// TIA Portal V20 export
FUNCTION_BLOCK "CallProcessCount"   // FB2, LAD
// stored: MemoryReserve 100, SetENOAutomatically false
   VAR
      statPulse { ExternalAccessible := 'False'; ExternalVisible := 'False'; ExternalWritable := 'False'} : Array[0..299] of Bool;
   END_VAR
   VAR_TEMP
      tempEnter : Bool;   // Enter the conditions for the count to increase.
   END_VAR
   VAR_TEMP   // added for the SCL form of the ladder/FBD networks
      _w1 : Bool;
   END_VAR
BEGIN

REGION Network 1: Production Data 1 Anode NG Parts
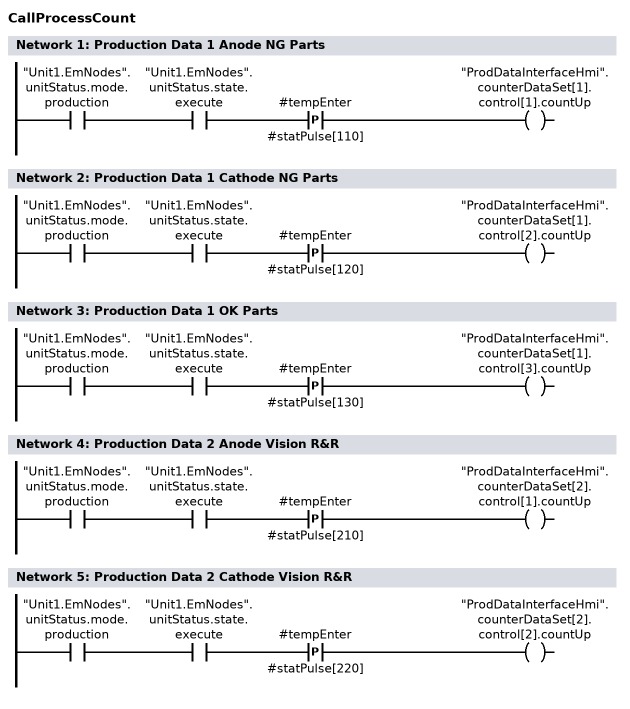
   RUNG wire#powerrail
      Contact( "Unit1.EmNodes".unitStatus.mode.production )
      Contact( "Unit1.EmNodes".unitStatus.state.execute )
      P_Contact(operand := #tempEnter, bit := #statPulse[110])
      Coil( "ProdDataInterfaceHmi".counterDataSet[1].control[1].countUp )
   END_RUNG
   // the same network as SCL:
   #_w1 := "Unit1.EmNodes".unitStatus.mode.production AND "Unit1.EmNodes".unitStatus.state.execute AND #tempEnter AND NOT #statPulse[110];   // rising edge of #tempEnter
   #statPulse[110] := #tempEnter;
   "ProdDataInterfaceHmi".counterDataSet[1].control[1].countUp := #_w1;
END_REGION

REGION Network 2: Production Data 1 Cathode NG Parts
   RUNG wire#powerrail
      Contact( "Unit1.EmNodes".unitStatus.mode.production )
      Contact( "Unit1.EmNodes".unitStatus.state.execute )
      P_Contact(operand := #tempEnter, bit := #statPulse[120])
      Coil( "ProdDataInterfaceHmi".counterDataSet[1].control[2].countUp )
   END_RUNG
   // the same network as SCL:
   #_w1 := "Unit1.EmNodes".unitStatus.mode.production AND "Unit1.EmNodes".unitStatus.state.execute AND #tempEnter AND NOT #statPulse[120];   // rising edge of #tempEnter
   #statPulse[120] := #tempEnter;
   "ProdDataInterfaceHmi".counterDataSet[1].control[2].countUp := #_w1;
END_REGION

REGION Network 3: Production Data 1 OK Parts
   RUNG wire#powerrail
      Contact( "Unit1.EmNodes".unitStatus.mode.production )
      Contact( "Unit1.EmNodes".unitStatus.state.execute )
      P_Contact(operand := #tempEnter, bit := #statPulse[130])
      Coil( "ProdDataInterfaceHmi".counterDataSet[1].control[3].countUp )
   END_RUNG
   // the same network as SCL:
   #_w1 := "Unit1.EmNodes".unitStatus.mode.production AND "Unit1.EmNodes".unitStatus.state.execute AND #tempEnter AND NOT #statPulse[130];   // rising edge of #tempEnter
   #statPulse[130] := #tempEnter;
   "ProdDataInterfaceHmi".counterDataSet[1].control[3].countUp := #_w1;
END_REGION

REGION Network 4: Production Data 2 Anode Vision R&R
   RUNG wire#powerrail
      Contact( "Unit1.EmNodes".unitStatus.mode.production )
      Contact( "Unit1.EmNodes".unitStatus.state.execute )
      P_Contact(operand := #tempEnter, bit := #statPulse[210])
      Coil( "ProdDataInterfaceHmi".counterDataSet[2].control[1].countUp )
   END_RUNG
   // the same network as SCL:
   #_w1 := "Unit1.EmNodes".unitStatus.mode.production AND "Unit1.EmNodes".unitStatus.state.execute AND #tempEnter AND NOT #statPulse[210];   // rising edge of #tempEnter
   #statPulse[210] := #tempEnter;
   "ProdDataInterfaceHmi".counterDataSet[2].control[1].countUp := #_w1;
END_REGION

REGION Network 5: Production Data 2 Cathode Vision R&R
   RUNG wire#powerrail
      Contact( "Unit1.EmNodes".unitStatus.mode.production )
      Contact( "Unit1.EmNodes".unitStatus.state.execute )
      P_Contact(operand := #tempEnter, bit := #statPulse[220])
      Coil( "ProdDataInterfaceHmi".counterDataSet[2].control[2].countUp )
   END_RUNG
   // the same network as SCL:
   #_w1 := "Unit1.EmNodes".unitStatus.mode.production AND "Unit1.EmNodes".unitStatus.state.execute AND #tempEnter AND NOT #statPulse[220];   // rising edge of #tempEnter
   #statPulse[220] := #tempEnter;
   "ProdDataInterfaceHmi".counterDataSet[2].control[2].countUp := #_w1;
END_REGION
END_FUNCTION_BLOCK
